PROGRAM PLC_SW1
VAR_INPUT
	nSocketType:UINT:=1;// socket 类型; 0 表示 server; 1 表示 client;
	sTerminalName:STRING;// 通讯对方名称 自定义
	sHost:STRING(20):='127.0.0.1';// 通讯IP地址; server时表示本地host; client时表示远程host
	nPort:UDINT:=8900;// 通讯端口号;
	bEnable:BOOL:=TRUE;// 通讯启用\禁用连接
	sSendSuffix:STRING:='';//此处可统一添加发送后缀字符 $R$N
	nQueueInterval:UDINT:=50;// 发送队列时间间隔 单位ms
	logHandleArray:ARRAY [1..5] OF POINTER TO printLogModule_EX;// log 操作 handle 数组
	logHandleArrayLength:UINT:=0;// log 操作 handle 数组长度, 不超过5
	enHeartBeat:BOOL;// 启用心跳包命令
	cmdHeartBeat:DINT;// 心跳包命令
	
	ResignOK:BOOL;
	Stop:BOOL;
	Aoi1Result:BOOL;
	stopmsg:WSTRING;
END_VAR
VAR_OUTPUT
	bSendCondition	:BOOL;//可发送条件
	bSocketConnected:BOOL;//连接状态
	
	Stopppp:BOOL:=FALSE;;
END_VAR
VAR CONSTANT
	cNumBegin		:DINT:=1;
	cNumEnd			:DINT:=100;
END_VAR
VAR
	sendDataArray	:ARRAY [cNumBegin..cNumEnd] OF struct_Tester;
	length			:DINT:=0;
	endPoint		:DINT:=cNumBegin;
	sendPoint		:DINT:=cNumBegin;
	passMax			:BOOL;
	popupSendData	:struct_Tester;
	//popup
	popupStep		:UINT:=0;
	popupTON1		:TON;
	popupTON2		:TON;
	iPopup			:DINT:=0;
	_PopupLength	:DINT:=0;
END_VAR
VAR
	tcpipClient					:tcpipClientModule_EX;
	tcpipServer					:tcpipServerModule_EX;////定义服务器对象
	
	tcpipSendDataBuff_Server	:ST_TCPIP_DATA_STRUCT_ALC;//发送数据 Buff server
	tcpipSendDataBuff_Client	:ST_TCPIP_DATA_STRUCT_ALC;//发送数据 Buff client
	
	tcpipSendDataClear			:ST_TCPIP_DATA_STRUCT_ALC;//发送数据 清空
	tcpipSendData				:ST_TCPIP_DATA_STRUCT_ALC;//发送数据
	
	tcpipRecDataBuff_Server		:ST_TCPIP_DATA_STRUCT_ALC;//已接收数据 Buff server
	tcpipRecDataBuff_Client		:ST_TCPIP_DATA_STRUCT_ALC;//已接收数据 Buff client
	
	tcpipRecDataClear			:ST_TCPIP_DATA_STRUCT_ALC;//已接收数据 清空
	tcpipRecData				:ST_TCPIP_DATA_STRUCT_ALC;//已接收数据
	
	tcpConnectR_Trig			:R_Trig;//初始连接上升沿
	tcpConnectF_Trig			:F_Trig;//初始连接下降沿
	registerStep				:UDINT;//ALC注册控制步
	registerTON					:TON;//ALC注册延时
	
	logHandleArray_index		:UINT:=1;
END_VAR
VAR
	(*
	bTrig_Version:BOOL;
	rTrig_Version:R_TRIG;
	*)
END_VAR


CASE nSocketType OF
0://TCPIP server
	tcpipServer(
		sSrvNetId:= , 
		sLocalHost:=sHost , 
		nLocalPort:=nPort , 
		bStartConnect:=bEnable , 
		tcpipSDataLen:=SIZEOF(tcpipSendDataBuff_Server) , 
		tcpipSData:=ADR(tcpipSendDataBuff_Server) , 
		bSend:= , 
		tcpipRecDataLen:=SIZEOF(tcpipRecDataBuff_Server) , 
		tcpipRecData:=ADR(tcpipRecDataBuff_Server) , 
		bAccepted=> , 
		bSendBusy=> , 
		bRecData=> );
	bSendCondition:=tcpipServer.bAccepted AND NOT tcpipServer.bSendBusy;
	//TCPIP连接
	bSocketConnected:=tcpipServer.bAccepted;
	IF NOT tcpipServer.bAccepted THEN
		length:=0;
		endPoint:=cNumBegin;
		sendPoint:=cNumBegin;
		passMax:=FALSE;
	END_IF
	tcpConnectR_Trig(CLK:=tcpipServer.bAccepted);
	tcpConnectF_Trig(CLK:=tcpipServer.bAccepted);

1://TCPIP client
	tcpipClient(
		sSrvNetId:= , 
		sRemoteHost:=sHost , 
		nRemotePort:=nPort , 
		bStartConnect:=bEnable , 
		tcpipSDataLen:=SIZEOF(tcpipSendDataBuff_Client) , 
		tcpipSData:=ADR(tcpipSendDataBuff_Client) , 
		bSend:= , 
		tcpipRecDataLen:=SIZEOF(tcpipRecDataBuff_Client) , 
		tcpipRecData:=ADR(tcpipRecDataBuff_Client) , 
		bConnected=> , 
		bSendBusy=> , 
		bRecData=> );
	bSendCondition:=tcpipClient.bConnected AND NOT tcpipClient.bSendBusy;
	//TCPIP连接
	bSocketConnected:=tcpipClient.bConnected;
	IF NOT tcpipClient.bConnected THEN
		length:=0;
		endPoint:=cNumBegin;
		sendPoint:=cNumBegin;
		passMax:=FALSE;
	END_IF
	tcpConnectR_Trig(CLK:=tcpipClient.bConnected);
	tcpConnectF_Trig(CLK:=tcpipClient.bConnected);
END_CASE

IF tcpConnectR_Trig.Q THEN
	FOR logHandleArray_index:=1 TO logHandleArrayLength DO
		logHandleArray[logHandleArray_index]^.append(CONCAT(sTerminalName, ' has been connected'));
	END_FOR
	registerStep:=10;
END_IF
IF tcpConnectF_Trig.Q THEN
	FOR logHandleArray_index:=1 TO logHandleArrayLength DO
		logHandleArray[logHandleArray_index]^.append(CONCAT(sTerminalName, ' has been disconnected'));
	END_FOR
	registerStep:=0;
END_IF
//数据接收处理
CASE nSocketType OF
0://TCPIP server
	IF tcpipServer.bRecData THEN
		tcpipRecData:=tcpipRecDataBuff_Server;//buff转存
		tcpipRecDataBuff_Server:=tcpipRecDataClear;//转存之后清空buff
		dataProcessing();
	END_IF
1://TCPIP client
	IF tcpipClient.bRecData THEN
		tcpipRecData:=tcpipRecDataBuff_Client;//buff转存
		tcpipRecDataBuff_Client:=tcpipRecDataClear;//转存之后清空buff
		dataProcessing();
	END_IF
END_CASE


popup();

CASE registerStep OF
0:
	//Ready
10:
	registerStep:=0;
// 心跳包
20:
	IF NOT enHeartBeat THEN
		registerStep:=0;
	ELSE
		registerStep:=registerStep+10;
	END_IF
30:
	registerTON(IN:=FALSE);
	appendSend(1,0,cmdHeartBeat,0.0,0.0,0.0,0.0,0.0,0,'');
	registerStep:=registerStep+10;
40:
	registerTON(IN:=NOT registerTON.Q,PT:=T#3S);
	IF registerTON.Q THEN
		registerTON(IN:=FALSE);
		registerStep:=30;
	END_IF
END_CASE

Manual();

METHOD appendSend : BOOL
VAR_INPUT
	channel		:DINT;
	msgType		:DINT:=0;
	funCode		:DINT;
	value1		:REAL:=0;
	value2		:REAL:=0;
	value3		:REAL:=0;
	value4		:REAL:=0;
	value5		:REAL:=0;
	errID		:LINT:=0;
	str			:STRING(g_nMaxByte_Client):='';
END_VAR

sendDataArray[endPoint].channel:=channel;
sendDataArray[endPoint].msgType:=msgType;
sendDataArray[endPoint].funCode:=funCode;
sendDataArray[endPoint].msgType:=msgType;
sendDataArray[endPoint].value1:=value1;
sendDataArray[endPoint].value2:=value2;
sendDataArray[endPoint].value3:=value3;
sendDataArray[endPoint].value4:=value4;
sendDataArray[endPoint].value5:=value5;
sendDataArray[endPoint].errID:=errID;
sendDataArray[endPoint].str:=str;

endPoint:=endPoint+1;
IF endPoint>(cNumEnd-1) THEN
	endPoint:=1;
	passMax:=TRUE;
END_IF
END_METHOD

METHOD dataProcessing : BOOL
VAR_INPUT
END_VAR
VAR
	i_CGResult:INT;
	i_HResult:INT;
END_VAR
FOR logHandleArray_index:=1 TO logHandleArrayLength DO
	CASE nSocketType OF
	0://TCPIP server
		IF enHeartBeat AND tcpipRecData.funCode=cmdHeartBeat THEN// 不打印心跳包命令
			EXIT;
		END_IF
		logHandleArray[logHandleArray_index]^.append(CONCAT(CONCAT(CONCAT('Recevie From ', sTerminalName), ' -- '),ALCData2String(tcpipRecData)));
	1://TCPIP client
		IF enHeartBeat AND tcpipRecData.funCode=cmdHeartBeat THEN// 不打印心跳包命令
			EXIT;
		END_IF
		logHandleArray[logHandleArray_index]^.append(CONCAT(CONCAT(CONCAT('Recevie From ', sTerminalName), ' -- '),ALCData2String(tcpipRecData)));
	END_CASE
END_FOR


CASE tcpipRecData.msgType OF
0://对方请求
	CASE tcpipRecData.funCode OF
	(*RotateStart_TM:
		gRotateStart_TM_Trig:=TRUE;
		gRotateStart_TM_SetVelo:=TO_LREAL(tcpipRecData.value1);
		Rotate_Start_POU.func_reset_status();
		Rotate_Start_POU.trigger:=TRUE;
		
		IF 0=tcpipRecData.errID THEN
			;
		ELSE
			;
		END_IF
		//appendSend(0,1,tcpipRecData.funCode,0.0,0.0,0.0,0.0,0.0,0,'');
	
	RotateStop_TM:
		IF 0=tcpipRecData.errID THEN
			;
		ELSE
			;
		END_IF
		//appendSend(0,1,tcpipRecData.funCode,0.0,0.0,0.0,0.0,0.0,0,'');
	*)
	END_CASE
1://对方响应
	CASE tcpipRecData.funCode OF
		1:
			//注册
			;
//			gRtnRegister := TRUE;
		
	END_CASE
END_CASE
END_METHOD

ACTION Manual:
(*
rTrig_Version(CLK:=bTrig_Version);
IF rTrig_Version.Q THEN
	appendSend(0,0,E_CmdID_SW.SW_GetVer,0.0,0.0,0.0,0.0,0.0,0,'');
END_IF
*)
END_ACTION

METHOD PRIVATE popup : BOOL
VAR_INPUT
END_VAR
CASE popupStep OF
0:
	IF (sendPoint<endPoint OR passMax) AND bSendCondition THEN
		popupSendData:=sendDataArray[sendPoint];
		sendData(popupSendData);//此处是调用信息发送
		popupStep:=10;
		sendPoint:=sendPoint+1;
		IF sendPoint>(cNumEnd-1) THEN
			sendPoint:=1;
			passMax:=FALSE;
		END_IF
	END_IF
10:
	popupTON2(IN:=NOT popupTON2.Q, PT:=T#2S);
	IF NOT bSendCondition OR popupTON2.Q THEN
		popupTON2(IN:=FALSE);
		popupStep:=11;
	END_IF
11:
	IF bSendCondition THEN
		popupStep:=12;
	END_IF
	popupTON1(IN:=FALSE);
12:
	//popupTON1(IN:=NOT popupTON1.Q,PT:=T#10MS);
	popupTON1(IN:=NOT popupTON1.Q,PT:=TO_TIME(nQueueInterval));
	IF popupTON1.Q THEN
		popupStep:=0;
	END_IF
END_CASE
END_METHOD


METHOD Register
VAR_INPUT
	nMachineType : INT;
END_VAR
//注册指令
appendSend(0,0,1, INT_TO_REAL(nMachineType),0.0,0.0,0.0,0.0,0,'');
END_METHOD

METHOD PRIVATE sendData : BOOL
VAR_INPUT
	dataStruct	:struct_Tester;
END_VAR
IF bSendCondition AND bEnable THEN
	tcpipSendData.channel	:=dataStruct.channel;
	tcpipSendData.msgType	:=dataStruct.msgType;
	tcpipSendData.funCode	:=dataStruct.funCode;
	tcpipSendData.value1	:=dataStruct.value1;
	tcpipSendData.value2	:=dataStruct.value2;
	tcpipSendData.value3	:=dataStruct.value3;
	tcpipSendData.value4	:=dataStruct.value4;
	tcpipSendData.value5	:=dataStruct.value5;
	tcpipSendData.errID		:=dataStruct.errID;
	tcpipSendData.str		:=tcpipServer.string2ASCII(dataStruct.str);
	
	CASE nSocketType OF
	0://TCPIP server
		tcpipSendDataBuff_Server:=tcpipSendData;
		tcpipSendData:=tcpipSendDataClear;	
		tcpipServer.bSend:=TRUE;
	1://TCPIP client
		tcpipSendDataBuff_Client:=tcpipSendData;
		tcpipSendData:=tcpipSendDataClear;	
		tcpipClient.bSend:=TRUE;
	END_CASE
	
	FOR logHandleArray_index:=1 TO logHandleArrayLength DO
		CASE nSocketType OF
		0://TCPIP server
			IF enHeartBeat AND dataStruct.funCode=cmdHeartBeat THEN// 不打印心跳包命令
				EXIT;
			END_IF
			logHandleArray[logHandleArray_index]^.append(CONCAT(CONCAT(CONCAT('Send To ', sTerminalName), ' -- '),ALCData2String(tcpipSendDataBuff_Server)));
		1://TCPIP client
			IF enHeartBeat AND dataStruct.funCode=cmdHeartBeat THEN// 不打印心跳包命令
				EXIT;
			END_IF
			logHandleArray[logHandleArray_index]^.append(CONCAT(CONCAT(CONCAT('Send To ', sTerminalName), ' -- '),ALCData2String(tcpipSendDataBuff_Client)));
		END_CASE
	END_FOR
END_IF
END_METHOD

END_PROGRAM

(* stored: Version 1.1.0.1, ProductVersion 3.1.4024.4
   POU PLC_SW1: Id {4cc1cd40-1206-4770-aded-6a81c6210c1a}, SpecialFunc None
   Folder CMD: Id {ac65ae50-0d77-45ca-b2b6-15cb70fc7ebb}
   Folder Recevie: Id {f5343d3b-801f-4793-b9e7-3bb0ccfff2b2}
   Folder Send: Id {2ed12d53-ffbb-4563-ab5c-b13057cdaea6}
   Folder Private: Id {728f8945-283e-4cb2-8271-ec9105d2ac58}
   Method appendSend: Id {cc1d9a5c-e9e8-4ba2-a195-465b176adc00}
   Method dataProcessing: Id {eceb49d1-8cc0-42da-98e2-c68c4bb1dce5}
   Action Manual: Id {fef2cd56-2bc7-453c-8155-dc2642d8cbe3}
   Method popup: Id {e713b313-1f97-4583-bc28-3a379e883f0e}
   Method Register: Id {b820e63c-c532-4162-a9f7-aba16797da69}
   Method sendData: Id {aec5dae8-17e3-4aff-ae12-ab79082cf6ed} *)
